// TIA Portal V18 export
VAR_GLOBAL   // PLC tag table "11_CT-5"
   "iCT-5" AT %I8.3 : Bool;
   "oCT-5" AT %Q1.0 : Bool;
END_VAR
